TYPE ST_SCQ_6_0 :
(**************************************************************************************
 * 	Application		:	BoxControl Framework
 *	Revision		:	$Revision: 404529 $
 *	Revision date	:	$Date: 2018-04-23 08:21:38 +0200 (Mo., 23 Apr 2018) $
 *	Last changed by	:	$Author: b7bolm $
 *	URL				:	$URL: http://almscdc.swisslog.com/repo/SWPD/Development/BoxControlFramework/20_Release/trunk/01_Software/BCF/BCF/JumpStart/20_Product/10_App/11_Com/10_Lib/10_Conv/12_MFCS/11_SIS/01_DUTs/10_SIS_6_0/ST_SCQ_6_0.TcDUT $
 *
 *	Purpose			:	SCQ Structure
 *
 * ------------------------------------------------------------------------------------
 *	Copyright Swisslog [IP AG], Switzerland. All rights reserved.
 * 
 * ------------------------------------------------------------------------------------
 *	
 * 	Revision History: 
 *
 * 	VERSION			DATE			INITIALS			DESCRIPTION
 *	0.1				01.01.2001		swl					Example
 *
 **************************************************************************************)
STRUCT
	SubsystemName	: STRING(SIS_6_0.POSITION_STRINGLENGTH); // 12 Digit SIS Location MM-GGG-EEEE-FF-Z
	Code			: STRING(SIS_6_0.CONTROLCODE_STRINGLENGTH); // Control code 
	Variable		: STRING(SIS_6_0.CONTROLVARIABLE_STRINGLENGTH); // Control code variable 
	SystemTime		: STRING(SIS_6_0.TIMESTAMP_STRINGLENGTH); // 19 Digit TimeStamp YYYY-MM-DD-hh:mm:ss
END_STRUCT
END_TYPE

(* stored: Version 1.1.0.1, ProductVersion 3.1.4022.12
   DUT ST_SCQ_6_0: Id {d6d7b12d-6e4d-4f8f-815b-e56ed880c19f} *)
